// TIA Portal V20 export
TYPE "typeFDoorSignal"
// Safety status of door
// stored: Access Published, IsFailsafeCompliant true, Namespace Safety
   STRUCT
      reqDoorUnlock4 : Bool;   // Cmd Maint Door4 Open Request
      reqDoorUnlock5 : Bool;   // Cmd Maint Door5 Open Request
      reqDoorUnlock6 : Bool;   // Cmd Maint Door6 Open Request
      reqDoorUnlock7 : Bool;   // Cmd Maint Door7 Open Request
   END_STRUCT;
END_TYPE
